{attribute addProperty BoxType "KL2652-0050"}
{attribute addProperty Id "Channel_1Channel_B2ED953500Channel_2Channel_B2ED953500"}
{attribute addProperty CRC "3561416756"}
{attribute addProperty SizeInBites "0"}
{attribute addProperty SizeInBytes "0"}
TYPE KL_D446E834 :
STRUCT
	{attribute addProperty Name "Channel_1"}
	Channel_1 : Channel_B2ED9535;
	{attribute addProperty Name "Channel_2"}
	Channel_2 : Channel_B2ED9535;
END_STRUCT
END_TYPE

(* stored: Version 1.2.0.0, ProductVersion 3.1.4024.9
   DUT KL_D446E834: Id {1534e9ba-e527-4377-8880-2a95aac25e13} *)
